FUNCTION_BLOCK EcMasterDeviceState IMPLEMENTS IEcTask
VAR_INPUT
END_VAR
VAR_OUTPUT
END_VAR
VAR
	iState : INT;
	masterDeviceState : Tc2_EtherCAT.FB_EcGetMasterDevState;
	_execute: BOOL;
	_done: BOOL;
	_busy: BOOL;
	_error: BOOL;
	_netId: AMSNETID;
END_VAR

CASE iState OF
	0:
		IF _execute THEN
			_done := FALSE;
			_busy := TRUE;
			_error := FALSE;
			masterDeviceState.bExecute := TRUE;
			IF masterDeviceState.bBusy THEN
				iState := 10;
				_execute := false;
			END_IF
		END_IF
	10:
		IF NOT masterDeviceState.bBusy THEN
			IF NOT masterDeviceState.bError THEN
				_done := TRUE;
			ELSE
				_error := TRUE;
			END_IF
			_busy := FALSE;
			masterDeviceState.bExecute := FALSE;
			iState := 0;
		END_IF
END_CASE

masterDeviceState(sNetId := Tc2_System.F_CreateAmsNetId(nIds := NetId));

{warning 'add method implementation '}
METHOD Abort : BOOL
masterDeviceState.bExecute := FALSE;
_busy := FALSE;
_execute := FALSE;
Abort := TRUE;
iState := 0;
END_METHOD

{warning 'add property implementation'}
PROPERTY Busy : BOOL
GET
Busy := _busy;
END_GET
END_PROPERTY

{warning 'add property implementation'}
PROPERTY Done : BOOL
GET
Done := _done;
END_GET
END_PROPERTY

{warning 'add property implementation'}
PROPERTY Error : BOOL
GET
Error := _error;
END_GET
END_PROPERTY

{warning 'add method implementation '}
METHOD Execute : BOOL
IF NOT masterDeviceState.bBusy THEN
	Execute := _execute := true;
END_IF
END_METHOD

PROPERTY MasterDevState : word
GET
MasterDevState := masterDeviceState.nDevState;
END_GET
END_PROPERTY

{warning 'add property implementation'}
PROPERTY NetID : amsnetid
GET
NetID := _netId;
END_GET
SET
_netId := NetID;
END_SET
END_PROPERTY

END_FUNCTION_BLOCK

(* stored: Version 1.1.0.1, ProductVersion 3.1.4024.9
   POU EcMasterDeviceState: Id {bc133e4e-3e72-4aa8-8902-b5d51a594f13}, SpecialFunc None
   Method Abort: Id {46242914-fccb-406c-8400-8291d8a8f93a}
   Property Busy: Id {5da4c181-ee99-4d3d-9b37-dce34eb05670}
   Get Get: Id {11c23d11-caf2-448b-bde9-ae55574acdd1}
   Property Done: Id {a4dfbccd-de3f-4bc9-969a-77a04442b248}
   Get Get: Id {69db2e42-829a-4390-9e40-3e6ce7028cb2}
   Property Error: Id {0c40726e-946e-4761-8b5c-2a69114e131f}
   Get Get: Id {a94eccdc-261d-47ba-9dfd-07210315e423}
   Method Execute: Id {68d9020e-50a5-4b47-86e8-e12eafbc24a9}
   Property MasterDevState: Id {da9b7b29-89ba-4a34-97df-7393e4a67726}
   Get Get: Id {85e682a4-8915-42cb-a37d-1a9b41c7ff2d}
   Property NetID: Id {bbbbbe22-cad5-4b3e-93d4-5e5188de8cfe}
   Get Get: Id {57f2a269-6bdd-41ae-a31c-76cea7ba9793}
   Set Set: Id {dafb3a3e-2c6a-4b76-bf40-2bb3fe04ffd3} *)
